{attribute 'qualified_only'}
{attribute 'strict'}
TYPE eInternalTransitions :
(
	Configuring := 0,
	CleaningUp := 1,
	ShuttingDown := 2,
	Activating := 3,
	Deactivating := 4,
	ErrorProcessing := 5
);
END_TYPE

(* stored: Version 1.1.0.1, ProductVersion 3.1.4026.18
   DUT eInternalTransitions: Id {a1b2c3d4-5555-5555-5555-555555555555} *)
